FUNCTION_BLOCK fb_ele_controller
VAR_IN_OUT
	var_ref_ele : ref_ele_io;
END_VAR
VAR_INPUT
	in_flg_run : BOOL;
	in_var_moveMode : eP_eleMovemode;
	in_flg_pause : BOOL;
END_VAR
VAR_OUTPUT
	out_flg_run : BOOL;
	out_flg_busy: BOOL;
	out_flg_Done: BOOL;
	out_flg_error : BOOL;
END_VAR
VAR
	var_buf_eleMoveMode: eP_eleMoveMode;
	flg_eleADone: BOOL;
	flg_eleBDone: BOOL;
	flg_eleStopDone: BOOL;
	fbi_timOut: TON;
	fb_TON_delay: TON;
END_VAR
VAR // added by the converter: edge detectors and wires of the graphical bodies
    _rt1, _rt2, _rt3, _rt4 : R_TRIG;
    _ft1, _ft2 : F_TRIG;
    _w1, _w2, _w3, _w4, _w5, _w6, _w7, _w8 : BOOL;
END_VAR

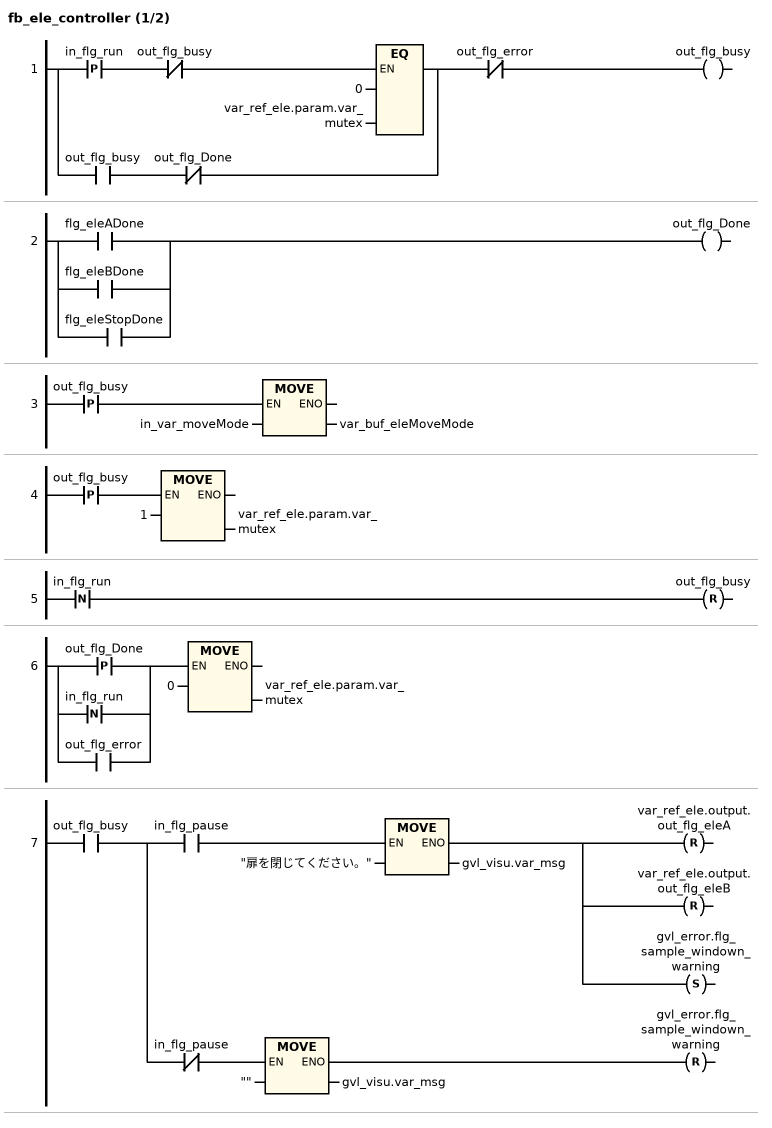
// NETWORK 1
_rt1(CLK := in_flg_run);
out_flg_busy := (_rt1.Q AND NOT out_flg_busy AND 0 = var_ref_ele.param.var_mutex OR out_flg_busy AND NOT out_flg_Done) AND NOT out_flg_error;

// NETWORK 2
out_flg_Done := flg_eleADone OR flg_eleBDone OR flg_eleStopDone;

// NETWORK 3
_rt2(CLK := out_flg_busy);
IF _rt2.Q THEN var_buf_eleMoveMode := in_var_moveMode; END_IF

// NETWORK 4
_rt3(CLK := out_flg_busy);
IF _rt3.Q THEN var_ref_ele.param.var_mutex := 1; END_IF

// NETWORK 5
_ft1(CLK := in_flg_run);
out_flg_busy R= _ft1.Q;

// NETWORK 6
_rt4(CLK := out_flg_Done);
_ft2(CLK := in_flg_run);
IF _rt4.Q OR _ft2.Q OR out_flg_error THEN var_ref_ele.param.var_mutex := 0; END_IF

// NETWORK 7
_w1 := out_flg_busy AND in_flg_pause;
IF _w1 THEN gvl_visu.var_msg := "扉を閉じてください。"; END_IF
var_ref_ele.output.out_flg_eleA R= _w1;
var_ref_ele.output.out_flg_eleB R= _w1;
gvl_error.flg_sample_windown_warning S= _w1;
_w2 := out_flg_busy AND NOT in_flg_pause;
IF _w2 THEN gvl_visu.var_msg := ""; END_IF
gvl_error.flg_sample_windown_warning R= _w2;

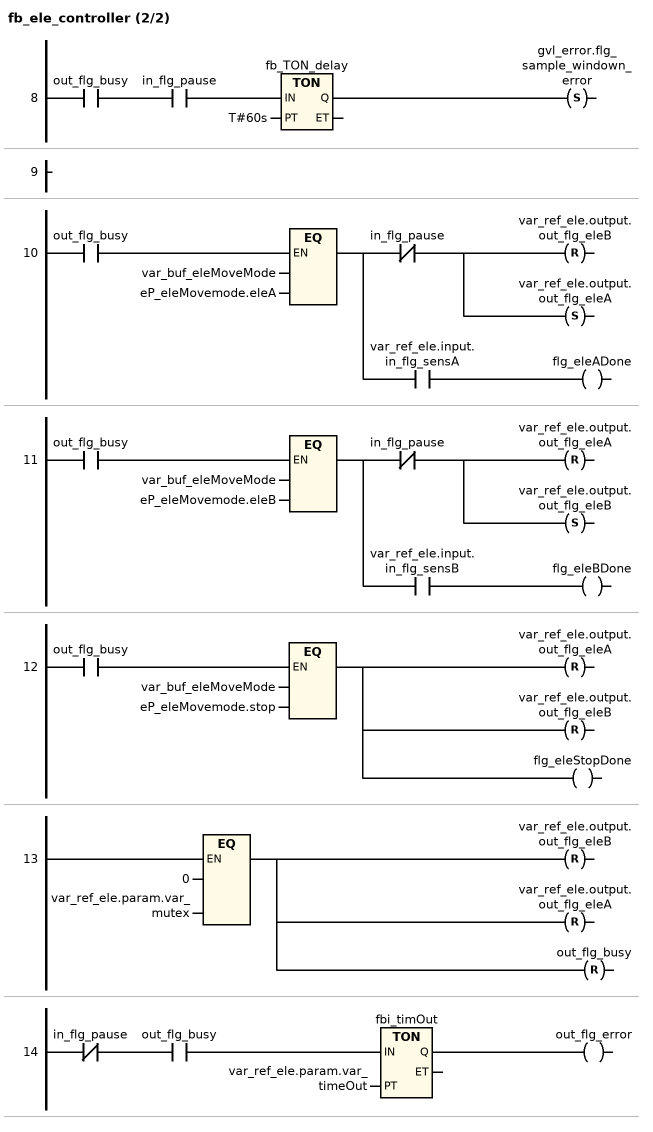
// NETWORK 8
fb_TON_delay(IN := out_flg_busy AND in_flg_pause, PT := T#60s); // TON
gvl_error.flg_sample_windown_error S= fb_TON_delay.Q;

// NETWORK 9

// NETWORK 10
_w3 := out_flg_busy AND var_buf_eleMoveMode = eP_eleMovemode.eleA;
_w4 := _w3 AND NOT in_flg_pause;
var_ref_ele.output.out_flg_eleB R= _w4;
var_ref_ele.output.out_flg_eleA S= _w4;
flg_eleADone := _w3 AND var_ref_ele.input.in_flg_sensA;

// NETWORK 11
_w5 := out_flg_busy AND var_buf_eleMoveMode = eP_eleMovemode.eleB;
_w6 := _w5 AND NOT in_flg_pause;
var_ref_ele.output.out_flg_eleA R= _w6;
var_ref_ele.output.out_flg_eleB S= _w6;
flg_eleBDone := _w5 AND var_ref_ele.input.in_flg_sensB;

// NETWORK 12
_w7 := out_flg_busy AND var_buf_eleMoveMode = eP_eleMovemode.stop;
var_ref_ele.output.out_flg_eleA R= _w7;
var_ref_ele.output.out_flg_eleB R= _w7;
flg_eleStopDone := _w7;

// NETWORK 13
_w8 := 0 = var_ref_ele.param.var_mutex;
var_ref_ele.output.out_flg_eleB R= _w8;
var_ref_ele.output.out_flg_eleA R= _w8;
out_flg_busy R= _w8;

// NETWORK 14
fbi_timOut(IN := NOT in_flg_pause AND out_flg_busy, PT := var_ref_ele.param.var_timeOut); // TON
out_flg_error := fbi_timOut.Q;

END_FUNCTION_BLOCK

(* stored: Version 1.1.0.1, ProductVersion 3.1.4024.11
   POU fb_ele_controller: Id {5d91ecdb-b24f-4c8c-993d-17ef02ccbaa9}, SpecialFunc None *)
